ABB RobotStudio station: VRT.rsstn

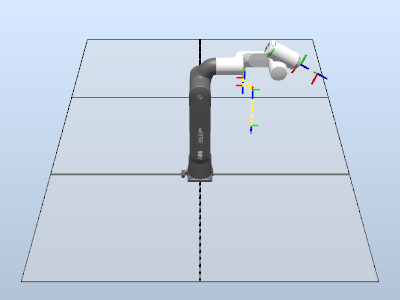
Station Station (saved by RobotStudio 22.3.10098.0)
Controller Virtual_RobotTeachIn
  mechanical unit ROB_1: CRB15000_5_95__02, 6 joints, base frame (0, 0, 0) mm
Layout (positions relative to the parent item):
  - CRB15000_5_95__02 [mechanism, from Robots\CRB15000_5_95__02.rslib] at (0, 0, 0) mm; joint values [0, 0, 0, 0, 0.5236, 0] (rad or m)
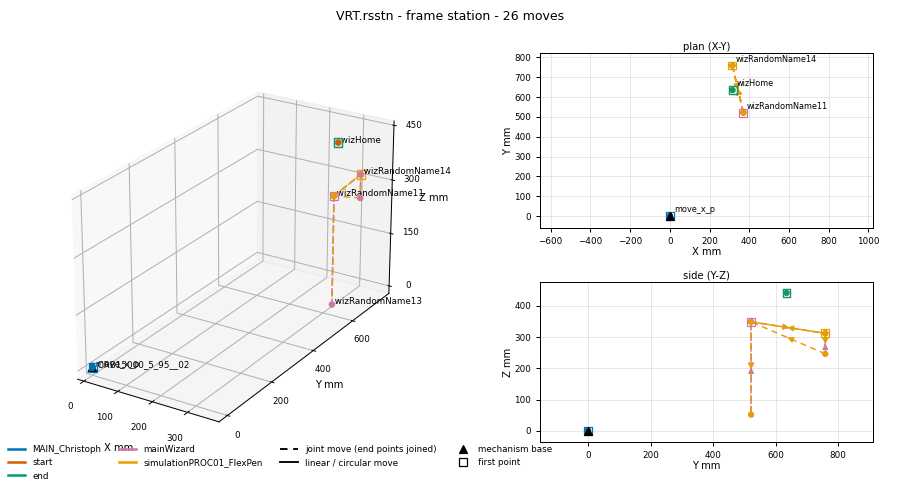
[picture p0: tool path of VRT.rsstn in frame station, 26 of 26 moves have a stored position in this frame; points joined in program order, loops and branches not executed]
Targets, tools, work objects and paths stored in the station, written as RAPID:
! task T_ROB1
MODULE MainModule
  TASK PERS tooldata tool1:=[TRUE,[[0,0,138],[0.980785,0,0,-0.19509]],[0.5,[0,0,0],[1,0,0,0],0,0,0]];
  TASK PERS tooldata tool_single_vacuum:=[TRUE,[[74.05,178.77,88.5],[0.5879378,-0.3928475,0.5879378,0.3928475]],[1,[0,0,0],[1,0,0,0],0,0,0]];
  LOCAL PERS wobjdata egm_wobj:=[FALSE,TRUE,"",[[0,1000,0],[1,0,0,0]],[[0,0,0],[1,0,0,0]]];
  CONST robtarget move_x_p:=[[1,0,0],[1,0,0,0],[0,0,0,0],[9E+09,9E+09,9E+09,9E+09,9E+09,9E+09]];
  CONST robtarget move_x_n:=[[-1,0,0],[1,0,0,0],[0,0,0,0],[9E+09,9E+09,9E+09,9E+09,9E+09,9E+09]];
  CONST robtarget move_y_p:=[[0,1,0],[1,0,0,0],[0,0,0,0],[9E+09,9E+09,9E+09,9E+09,9E+09,9E+09]];
  CONST robtarget move_y_n:=[[0,-1,0],[1,0,0,0],[0,0,0,0],[9E+09,9E+09,9E+09,9E+09,9E+09,9E+09]];
  CONST robtarget move_z_p:=[[0,0,1],[1,0,0,0],[0,0,0,0],[9E+09,9E+09,9E+09,9E+09,9E+09,9E+09]];
  CONST robtarget move_z_n:=[[0,0,-1],[1,0,0,0],[0,0,0,0],[9E+09,9E+09,9E+09,9E+09,9E+09,9E+09]];
  CONST robtarget move_rx_p:=[[0,0,0],[1,0,0,0],[0,0,0,0],[9E+09,9E+09,9E+09,9E+09,9E+09,9E+09]];
  CONST robtarget move_rx_n:=[[0,0,0],[1,0,0,0],[0,0,0,0],[9E+09,9E+09,9E+09,9E+09,9E+09,9E+09]];
  CONST robtarget move_ry_p:=[[0,0,0],[1,0,0,0],[0,0,0,0],[9E+09,9E+09,9E+09,9E+09,9E+09,9E+09]];
  CONST robtarget move_ry_n:=[[0,0,0],[1,0,0,0],[0,0,0,0],[9E+09,9E+09,9E+09,9E+09,9E+09,9E+09]];
  CONST robtarget move_rz_p:=[[0,0,0],[1,0,0,0],[0,0,0,0],[9E+09,9E+09,9E+09,9E+09,9E+09,9E+09]];
  CONST robtarget move_rz_n:=[[0,0,0],[1,0,0,0],[0,0,0,0],[9E+09,9E+09,9E+09,9E+09,9E+09,9E+09]];
  PROC MAIN_Christoph()
    MoveL move_x_p,v10,fine,tool0\WObj:=wobj0;
    MoveL move_x_n,v10,fine,tool0\WObj:=wobj0;
    MoveL move_y_p,v10,fine,tool0\WObj:=wobj0;
    MoveL move_y_n,v10,fine,tool0\WObj:=wobj0;
    MoveL move_z_p,v10,fine,tool0\WObj:=wobj0;
    MoveL move_z_n,v10,fine,tool0\WObj:=wobj0;
    MoveL move_rx_p,v10,fine,tool0\WObj:=wobj0;
    MoveL move_rx_n,v10,fine,tool0\WObj:=wobj0;
    MoveL move_ry_p,v10,fine,tool0\WObj:=wobj0;
    MoveL move_ry_n,v10,fine,tool0\WObj:=wobj0;
    MoveL move_rz_p,v10,fine,tool0\WObj:=wobj0;
    MoveL move_rz_n,v10,fine,tool0\WObj:=wobj0;
  ENDPROC
  PROC checkEgmConnection()
  ENDPROC
ENDMODULE

! task T_ROB1
MODULE module_MAIN
  PROC main()
  ENDPROC
ENDMODULE

! task T_ROB1
MODULE module_WIZARD
  PERS robtarget wizHome:=[[316.173339844,634.73046875,440.990356445],[0.0026821,0.007837469,0.999948502,0.005858082],[0,0,0,0],[9E+09,9E+09,9E+09,9E+09,9E+09,9E+09]];
  PERS robtarget wizRandomName11:=[[370.495269775,521.37487793,348.593353271],[0.003799025,0.701789558,0.712373674,-0.000882734],[0,-1,1,0],[9E+09,9E+09,9E+09,9E+09,9E+09,9E+09]];
  PERS robtarget wizRandomName13:=[[370.480529785,521.381530762,51.894950867],[0.003802514,0.708827674,0.705370903,-0.000862758],[0,-1,1,0],[9E+09,9E+09,9E+09,9E+09,9E+09,9E+09]];
  PERS robtarget wizRandomName14:=[[314.932128906,758.710083008,311.827056885],[0.002692041,0.007832407,0.999948382,0.005890123],[0,-1,0,0],[9E+09,9E+09,9E+09,9E+09,9E+09,9E+09]];
  PERS robtarget wizRandomName12:=[[314.909301758,758.708068848,246.256469727],[0.002686393,0.007815085,0.999948561,0.005880545],[0,-1,0,0],[9E+09,9E+09,9E+09,9E+09,9E+09,9E+09]];
  PERS robtarget wizRandomName03:=[[314.932128906,758.710083008,311.827056885],[0.002692041,0.007832407,0.999948382,0.005890123],[0,-1,0,0],[9E+09,9E+09,9E+09,9E+09,9E+09,9E+09]];
  PERS robtarget wizRandomName02:=[[370.495269775,521.37487793,348.593353271],[0.003799025,0.701789558,0.712373674,-0.000882734],[0,-1,1,0],[9E+09,9E+09,9E+09,9E+09,9E+09,9E+09]];
  PERS robtarget wizRandomName01:=[[314.909301758,758.708068848,246.256469727],[0.002686393,0.007815085,0.999948561,0.005880545],[0,-1,0,0],[9E+09,9E+09,9E+09,9E+09,9E+09,9E+09]];
  PERS robtarget wizRandomName04:=[[370.480529785,521.381530762,51.894950867],[0.003802514,0.708827674,0.705370903,-0.000862758],[0,-1,1,0],[9E+09,9E+09,9E+09,9E+09,9E+09,9E+09]];
  PROC start()
    MoveJ wizHome,v200,fine,tool0;
  ENDPROC
  PROC simulationPROC02_HoloLens2()
  ENDPROC
  PROC end()
    MoveJ wizHome,v200,fine,tool0;
  ENDPROC
  PROC mainWizard()
    start;
    MoveJ wizRandomName11,v100,fine,tool0;
    MoveJ wizRandomName13,v100,fine,tool0;
    MoveJ wizRandomName11,v100,fine,tool0;
    MoveJ wizRandomName14,v100,fine,tool0;
    MoveJ wizRandomName12,v100,fine,tool0;
    MoveJ wizRandomName14,v100,fine,tool0;
    end;
  ENDPROC
  PROC simulationPROC01_FlexPendant()
    start;
    MoveJ wizRandomName03,v100,fine,tool0;
    MoveJ wizRandomName02,v100,fine,tool0;
    MoveJ wizRandomName03,v100,fine,tool0;
    MoveJ wizRandomName01,v100,fine,tool0;
    MoveJ wizRandomName02,v100,fine,tool0;
    MoveJ wizRandomName04,v100,fine,tool0;
    end;
  ENDPROC
ENDMODULE

! task T_ROB1
MODULE module_mr19m010
  VAR triggdata trigg1;
  PROC main_mr19m010()
    WaitTime 0.5;
  ENDPROC
ENDMODULE

